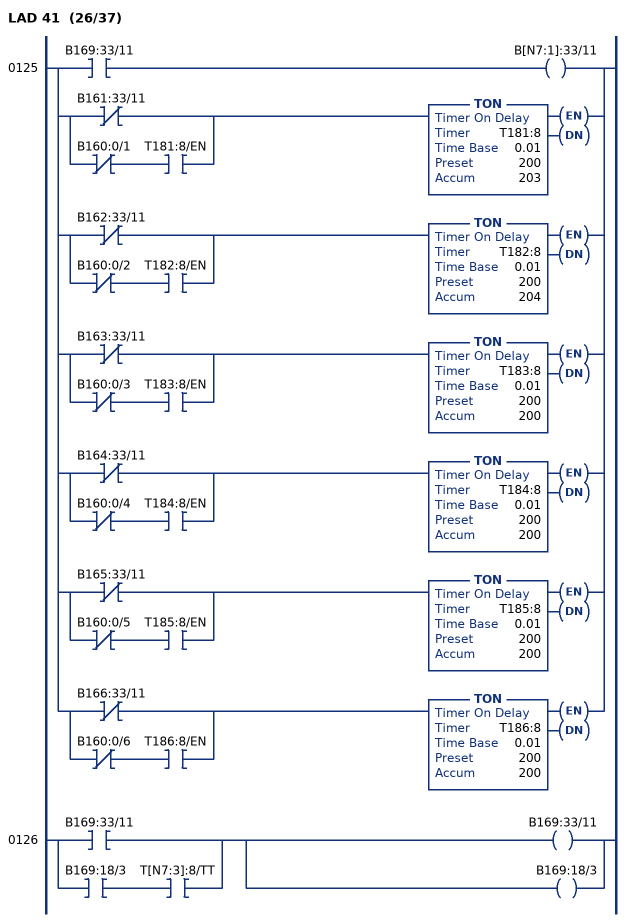
% Rung: 125 %
SOR BST XIC B169:33/11 OTE B[N7:1]:33/11 NXB BST XIO B161:33/11 NXB XIO B160:0/1 XIC T181:8/EN BND TON T181:8 0.01 200 203 NXB BST XIO B162:33/11 NXB XIO B160:0/2 XIC T182:8/EN BND TON T182:8 0.01 200 204 NXB BST XIO B163:33/11 NXB XIO B160:0/3 XIC T183:8/EN BND TON T183:8 0.01 200 200 NXB BST XIO B164:33/11 NXB XIO B160:0/4 XIC T184:8/EN BND TON T184:8 0.01 200 200 NXB BST XIO B165:33/11 NXB XIO B160:0/5 XIC T185:8/EN BND TON T185:8 0.01 200 200 NXB BST XIO B166:33/11 NXB XIO B160:0/6 XIC T186:8/EN BND TON T186:8 0.01 200 200 BND EOR
% Rung: 126 %
SOR BST XIC B169:33/11 NXB XIC B169:18/3 XIC T[N7:3]:8/TT BND BST OTE B169:33/11 NXB OTE B169:18/3 BND EOR

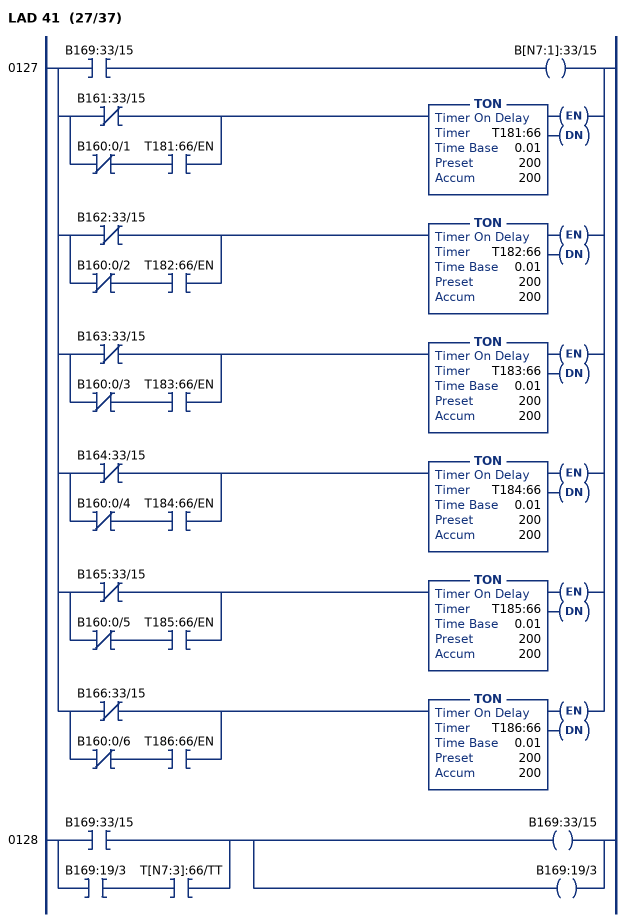
% Rung: 127 %
SOR BST XIC B169:33/15 OTE B[N7:1]:33/15 NXB BST XIO B161:33/15 NXB XIO B160:0/1 XIC T181:66/EN BND TON T181:66 0.01 200 200 NXB BST XIO B162:33/15 NXB XIO B160:0/2 XIC T182:66/EN BND TON T182:66 0.01 200 200 NXB BST XIO B163:33/15 NXB XIO B160:0/3 XIC T183:66/EN BND TON T183:66 0.01 200 200 NXB BST XIO B164:33/15 NXB XIO B160:0/4 XIC T184:66/EN BND TON T184:66 0.01 200 200 NXB BST XIO B165:33/15 NXB XIO B160:0/5 XIC T185:66/EN BND TON T185:66 0.01 200 200 NXB BST XIO B166:33/15 NXB XIO B160:0/6 XIC T186:66/EN BND TON T186:66 0.01 200 200 BND EOR
% Rung: 128 %
SOR BST XIC B169:33/15 NXB XIC B169:19/3 XIC T[N7:3]:66/TT BND BST OTE B169:33/15 NXB OTE B169:19/3 BND EOR

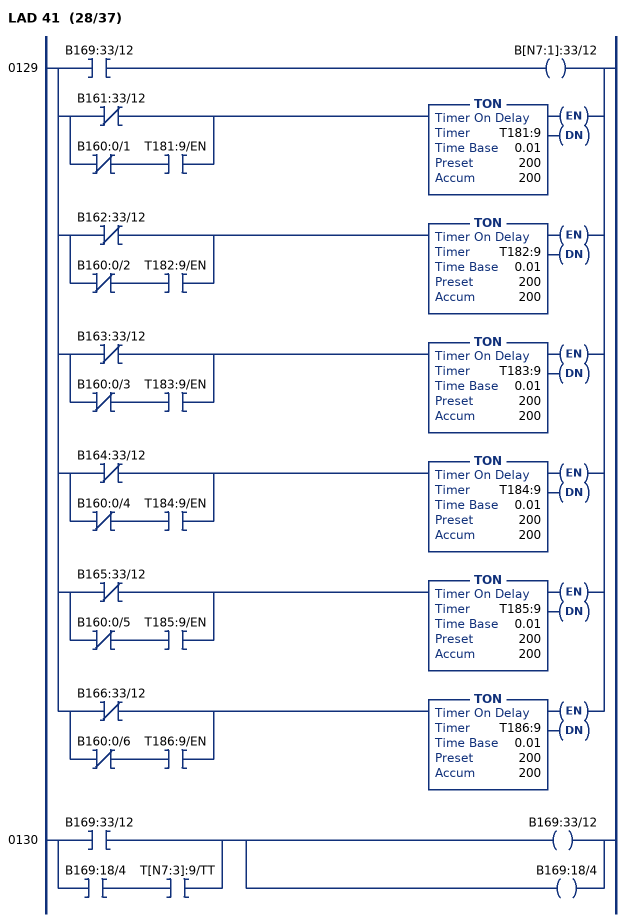
% Rung: 129 %
SOR BST XIC B169:33/12 OTE B[N7:1]:33/12 NXB BST XIO B161:33/12 NXB XIO B160:0/1 XIC T181:9/EN BND TON T181:9 0.01 200 200 NXB BST XIO B162:33/12 NXB XIO B160:0/2 XIC T182:9/EN BND TON T182:9 0.01 200 200 NXB BST XIO B163:33/12 NXB XIO B160:0/3 XIC T183:9/EN BND TON T183:9 0.01 200 200 NXB BST XIO B164:33/12 NXB XIO B160:0/4 XIC T184:9/EN BND TON T184:9 0.01 200 200 NXB BST XIO B165:33/12 NXB XIO B160:0/5 XIC T185:9/EN BND TON T185:9 0.01 200 200 NXB BST XIO B166:33/12 NXB XIO B160:0/6 XIC T186:9/EN BND TON T186:9 0.01 200 200 BND EOR
% Rung: 130 %
SOR BST XIC B169:33/12 NXB XIC B169:18/4 XIC T[N7:3]:9/TT BND BST OTE B169:33/12 NXB OTE B169:18/4 BND EOR

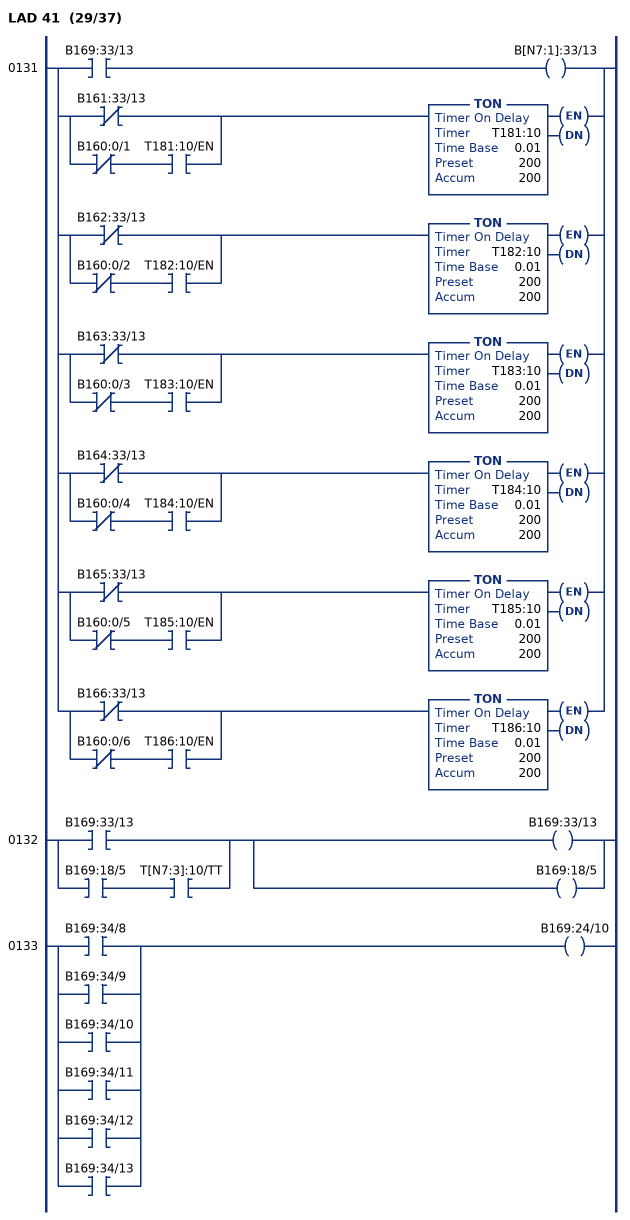
% Rung: 131 %
SOR BST XIC B169:33/13 OTE B[N7:1]:33/13 NXB BST XIO B161:33/13 NXB XIO B160:0/1 XIC T181:10/EN BND TON T181:10 0.01 200 200 NXB BST XIO B162:33/13 NXB XIO B160:0/2 XIC T182:10/EN BND TON T182:10 0.01 200 200 NXB BST XIO B163:33/13 NXB XIO B160:0/3 XIC T183:10/EN BND TON T183:10 0.01 200 200 NXB BST XIO B164:33/13 NXB XIO B160:0/4 XIC T184:10/EN BND TON T184:10 0.01 200 200 NXB BST XIO B165:33/13 NXB XIO B160:0/5 XIC T185:10/EN BND TON T185:10 0.01 200 200 NXB BST XIO B166:33/13 NXB XIO B160:0/6 XIC T186:10/EN BND TON T186:10 0.01 200 200 BND EOR
% Rung: 132 %
SOR BST XIC B169:33/13 NXB XIC B169:18/5 XIC T[N7:3]:10/TT BND BST OTE B169:33/13 NXB OTE B169:18/5 BND EOR
% Rung: 133 %
SOR BST XIC B169:34/8 NXB XIC B169:34/9 NXB XIC B169:34/10 NXB XIC B169:34/11 NXB XIC B169:34/12 NXB XIC B169:34/13 BND OTE B169:24/10 EOR

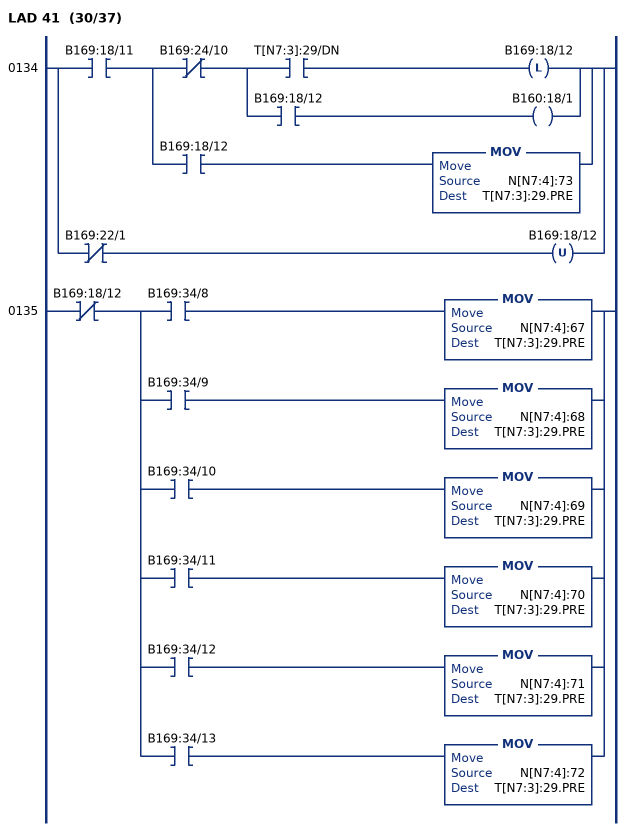
% Rung: 134 %
SOR BST XIC B169:18/11 BST XIO B169:24/10 BST XIC T[N7:3]:29/DN OTL B169:18/12 NXB XIC B169:18/12 OTE B160:18/1 BND NXB XIC B169:18/12 MOV N[N7:4]:73 T[N7:3]:29.PRE BND NXB XIO B169:22/1 OTU B169:18/12 BND EOR
% Rung: 135 %
SOR XIO B169:18/12 BST XIC B169:34/8 MOV N[N7:4]:67 T[N7:3]:29.PRE NXB XIC B169:34/9 MOV N[N7:4]:68 T[N7:3]:29.PRE NXB XIC B169:34/10 MOV N[N7:4]:69 T[N7:3]:29.PRE NXB XIC B169:34/11 MOV N[N7:4]:70 T[N7:3]:29.PRE NXB XIC B169:34/12 MOV N[N7:4]:71 T[N7:3]:29.PRE NXB XIC B169:34/13 MOV N[N7:4]:72 T[N7:3]:29.PRE BND EOR

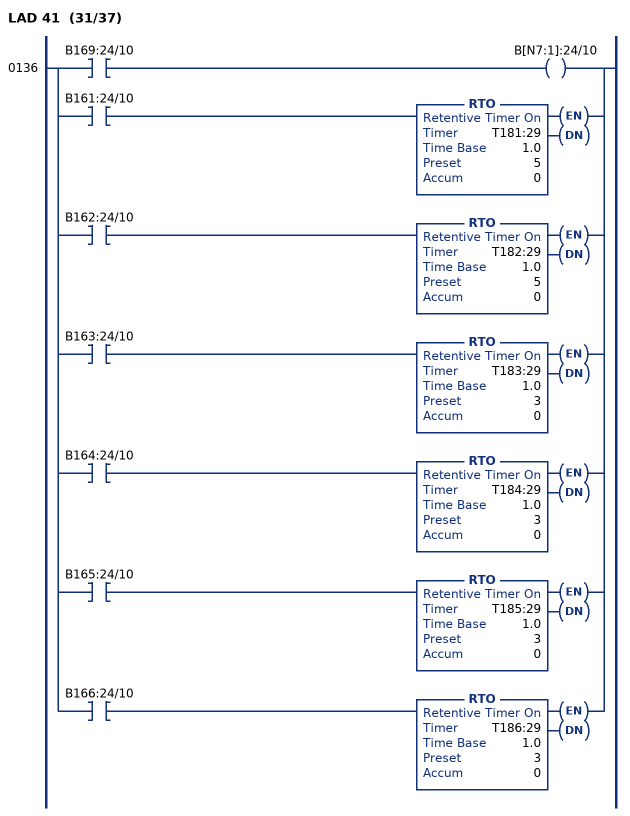
% Rung: 136 %
SOR BST XIC B169:24/10 OTE B[N7:1]:24/10 NXB XIC B161:24/10 RTO T181:29 1.0 5 0 NXB XIC B162:24/10 RTO T182:29 1.0 5 0 NXB XIC B163:24/10 RTO T183:29 1.0 3 0 NXB XIC B164:24/10 RTO T184:29 1.0 3 0 NXB XIC B165:24/10 RTO T185:29 1.0 3 0 NXB XIC B166:24/10 RTO T186:29 1.0 3 0 BND EOR

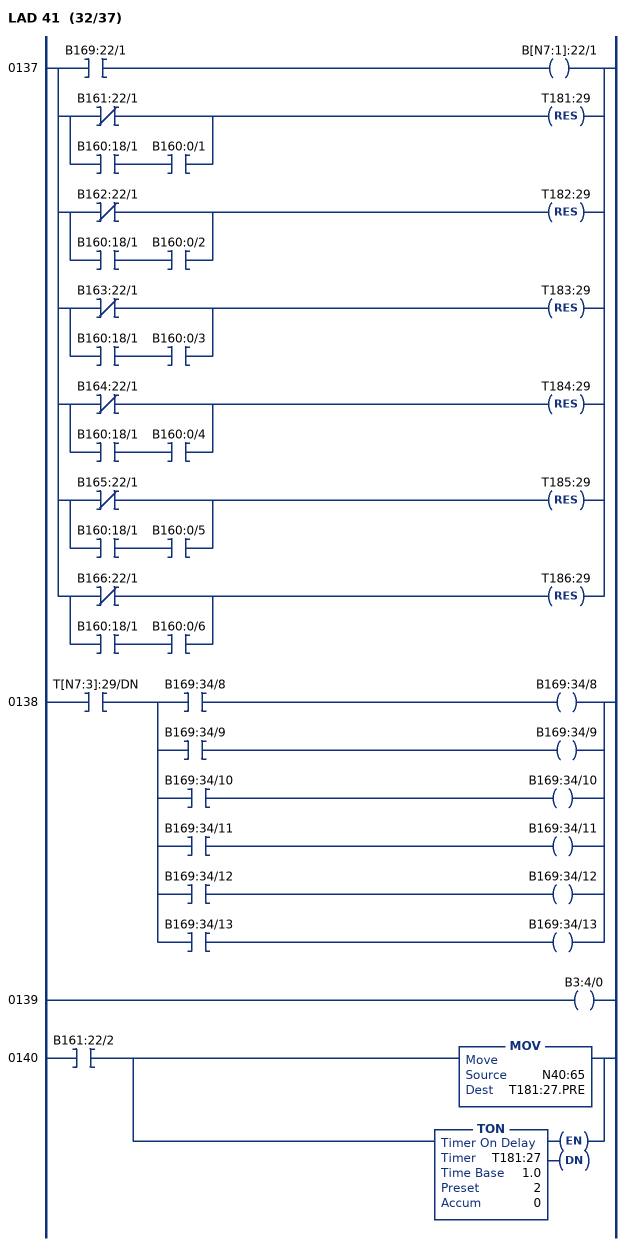
% Rung: 137 %
SOR BST XIC B169:22/1 OTE B[N7:1]:22/1 NXB BST XIO B161:22/1 NXB XIC B160:18/1 XIC B160:0/1 BND RES T181:29 NXB BST XIO B162:22/1 NXB XIC B160:18/1 XIC B160:0/2 BND RES T182:29 NXB BST XIO B163:22/1 NXB XIC B160:18/1 XIC B160:0/3 BND RES T183:29 NXB BST XIO B164:22/1 NXB XIC B160:18/1 XIC B160:0/4 BND RES T184:29 NXB BST XIO B165:22/1 NXB XIC B160:18/1 XIC B160:0/5 BND RES T185:29 NXB BST XIO B166:22/1 NXB XIC B160:18/1 XIC B160:0/6 BND RES T186:29 BND EOR
% Rung: 138 %
SOR XIC T[N7:3]:29/DN BST XIC B169:34/8 OTE B169:34/8 NXB XIC B169:34/9 OTE B169:34/9 NXB XIC B169:34/10 OTE B169:34/10 NXB XIC B169:34/11 OTE B169:34/11 NXB XIC B169:34/12 OTE B169:34/12 NXB XIC B169:34/13 OTE B169:34/13 BND EOR
% Rung: 139 %
SOR OTE B3:4/0 EOR
% Rung: 140 %
SOR XIC B161:22/2 BST MOV N40:65 T181:27.PRE NXB TON T181:27 1.0 2 0 BND EOR

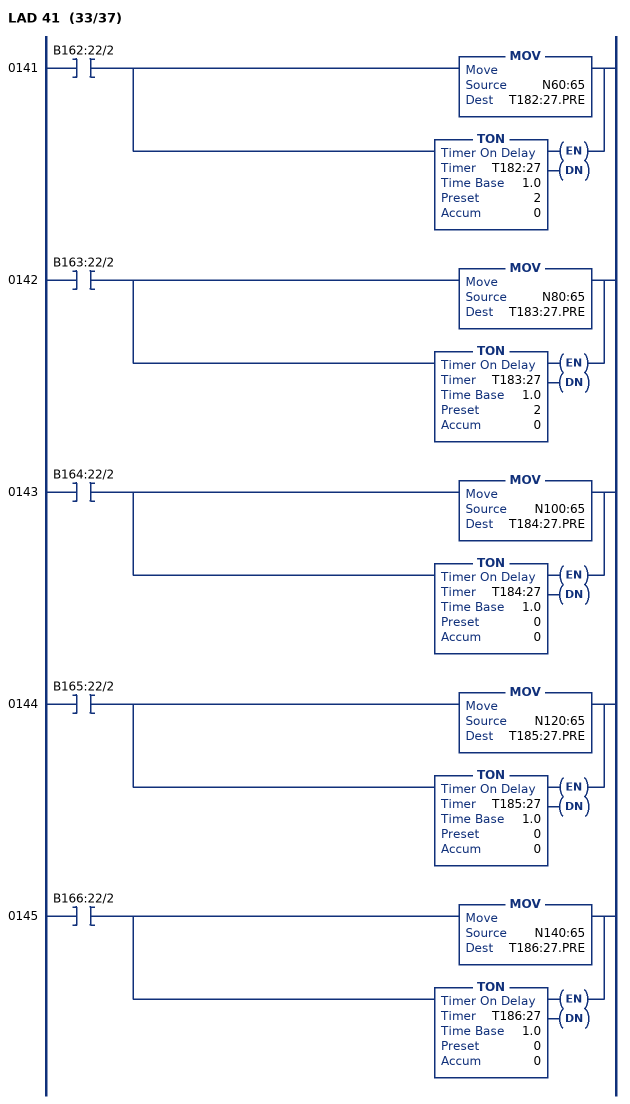
% Rung: 141 %
SOR XIC B162:22/2 BST MOV N60:65 T182:27.PRE NXB TON T182:27 1.0 2 0 BND EOR
% Rung: 142 %
SOR XIC B163:22/2 BST MOV N80:65 T183:27.PRE NXB TON T183:27 1.0 2 0 BND EOR
% Rung: 143 %
SOR XIC B164:22/2 BST MOV N100:65 T184:27.PRE NXB TON T184:27 1.0 0 0 BND EOR
% Rung: 144 %
SOR XIC B165:22/2 BST MOV N120:65 T185:27.PRE NXB TON T185:27 1.0 0 0 BND EOR
% Rung: 145 %
SOR XIC B166:22/2 BST MOV N140:65 T186:27.PRE NXB TON T186:27 1.0 0 0 BND EOR

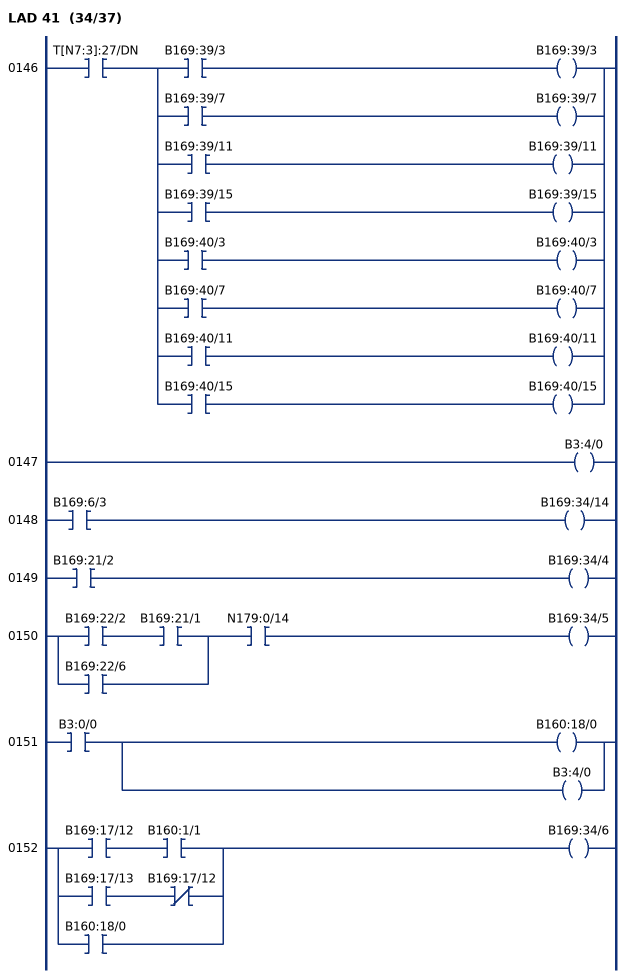
% Rung: 146 %
SOR XIC T[N7:3]:27/DN BST XIC B169:39/3 OTE B169:39/3 NXB XIC B169:39/7 OTE B169:39/7 NXB XIC B169:39/11 OTE B169:39/11 NXB XIC B169:39/15 OTE B169:39/15 NXB XIC B169:40/3 OTE B169:40/3 NXB XIC B169:40/7 OTE B169:40/7 NXB XIC B169:40/11 OTE B169:40/11 NXB XIC B169:40/15 OTE B169:40/15 BND EOR
% Rung: 147 %
SOR OTE B3:4/0 EOR
% Rung: 148 %
SOR XIC B169:6/3 OTE B169:34/14 EOR
% Rung: 149 %
SOR XIC B169:21/2 OTE B169:34/4 EOR
% Rung: 150 %
SOR BST XIC B169:22/2 XIC B169:21/1 NXB XIC B169:22/6 BND XIC N179:0/14 OTE B169:34/5 EOR
% Rung: 151 %
SOR XIC B3:0/0 BST OTE B160:18/0 NXB OTE B3:4/0 BND EOR
% Rung: 152 %
SOR BST XIC B169:17/12 XIC B160:1/1 NXB XIC B169:17/13 XIO B169:17/12 NXB XIC B160:18/0 BND OTE B169:34/6 EOR

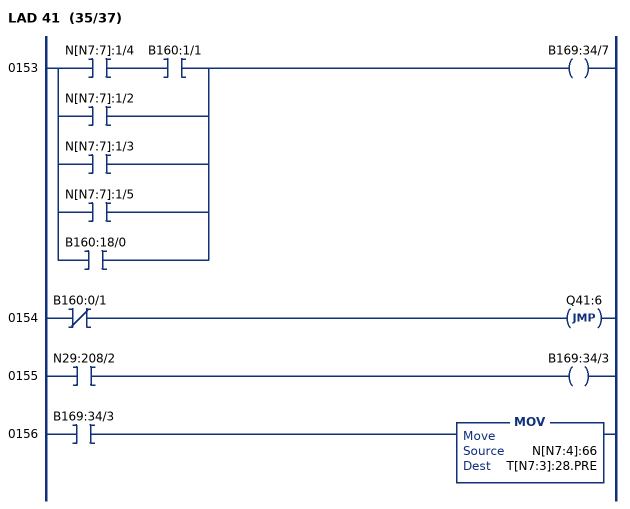
% Rung: 153 %
SOR BST XIC N[N7:7]:1/4 XIC B160:1/1 NXB XIC N[N7:7]:1/2 NXB XIC N[N7:7]:1/3 NXB XIC N[N7:7]:1/5 NXB XIC B160:18/0 BND OTE B169:34/7 EOR
% Rung: 154 %
SOR XIO B160:0/1 JMP Q41:6 EOR
% Rung: 155 %
SOR XIC N29:208/2 OTE B169:34/3 EOR
% Rung: 156 %
SOR XIC B169:34/3 MOV N[N7:4]:66 T[N7:3]:28.PRE EOR

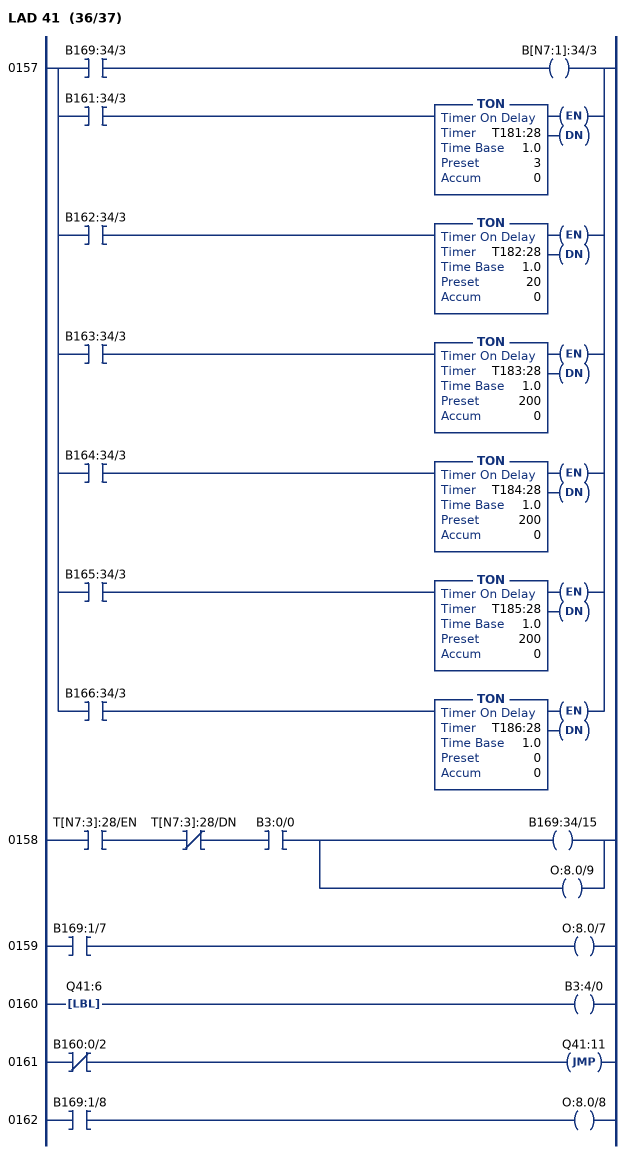
% Rung: 157 %
SOR BST XIC B169:34/3 OTE B[N7:1]:34/3 NXB XIC B161:34/3 TON T181:28 1.0 3 0 NXB XIC B162:34/3 TON T182:28 1.0 20 0 NXB XIC B163:34/3 TON T183:28 1.0 200 0 NXB XIC B164:34/3 TON T184:28 1.0 200 0 NXB XIC B165:34/3 TON T185:28 1.0 200 0 NXB XIC B166:34/3 TON T186:28 1.0 0 0 BND EOR
% Rung: 158 %
SOR XIC T[N7:3]:28/EN XIO T[N7:3]:28/DN XIC B3:0/0 BST OTE B169:34/15 NXB OTE O:8.0/9 BND EOR
% Rung: 159 %
SOR XIC B169:1/7 OTE O:8.0/7 EOR
% Rung: 160 %
SOR LBL Q41:6 OTE B3:4/0 EOR
% Rung: 161 %
SOR XIO B160:0/2 JMP Q41:11 EOR
% Rung: 162 %
SOR XIC B169:1/8 OTE O:8.0/8 EOR

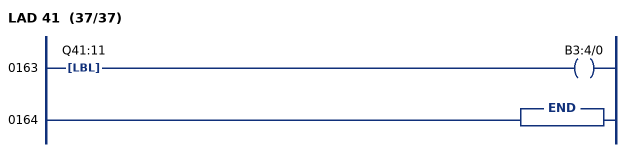
% Rung: 163 %
SOR LBL Q41:11 OTE B3:4/0 EOR
% Rung: 164 %
SOR END EOR

LADDER 42
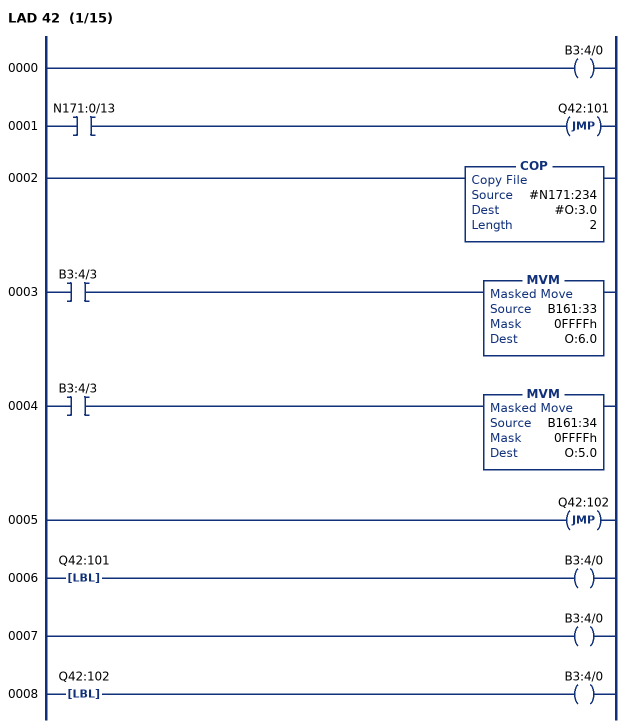
% Rung: 0 %
SOR OTE B3:4/0 EOR
% Rung: 1 %
SOR XIC N171:0/13 JMP Q42:101 EOR
% Rung: 2 %
SOR COP #N171:234 #O:3.0 2 EOR
% Rung: 3 %
SOR XIC B3:4/3 MVM B161:33 0FFFFh O:6.0 EOR
% Rung: 4 %
SOR XIC B3:4/3 MVM B161:34 0FFFFh O:5.0 EOR
% Rung: 5 %
SOR JMP Q42:102 EOR
% Rung: 6 %
SOR LBL Q42:101 OTE B3:4/0 EOR
% Rung: 7 %
SOR OTE B3:4/0 EOR
% Rung: 8 %
SOR LBL Q42:102 OTE B3:4/0 EOR

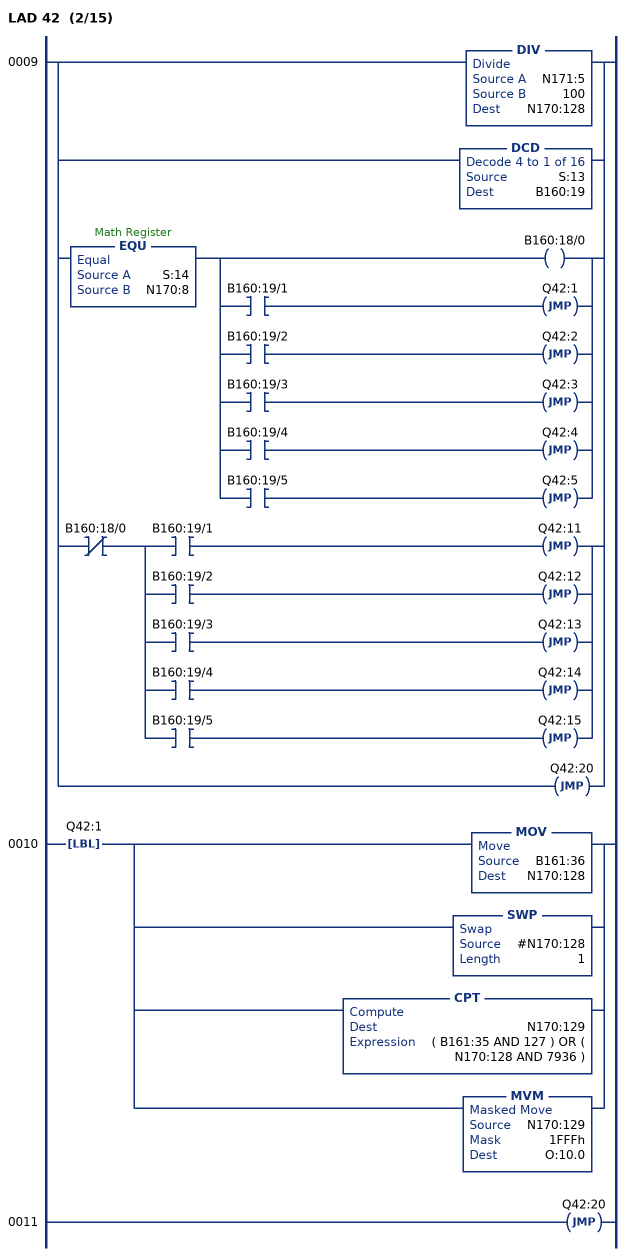
% Rung: 9 %
SOR BST DIV N171:5 100 N170:128 NXB DCD S:13 B160:19 NXB EQU S:14 N170:8 BST OTE B160:18/0 NXB XIC B160:19/1 JMP Q42:1 NXB XIC B160:19/2 JMP Q42:2 NXB XIC B160:19/3 JMP Q42:3 NXB XIC B160:19/4 JMP Q42:4 NXB XIC B160:19/5 JMP Q42:5 BND NXB XIO B160:18/0 BST XIC B160:19/1 JMP Q42:11 NXB XIC B160:19/2 JMP Q42:12 NXB XIC B160:19/3 JMP Q42:13 NXB XIC B160:19/4 JMP Q42:14 NXB XIC B160:19/5 JMP Q42:15 BND NXB JMP Q42:20 BND EOR
%   S:13  "Math Register" %
%   S:14  "Math Register" %
% Rung: 10 %
SOR LBL Q42:1 BST MOV B161:36 N170:128 NXB SWP #N170:128 1 NXB CPT N170:129 " ( B161:35 AND 127 ) OR ( N170:128 AND 7936 ) " NXB MVM N170:129 1FFFh O:10.0 BND EOR
% Rung: 11 %
SOR JMP Q42:20 EOR

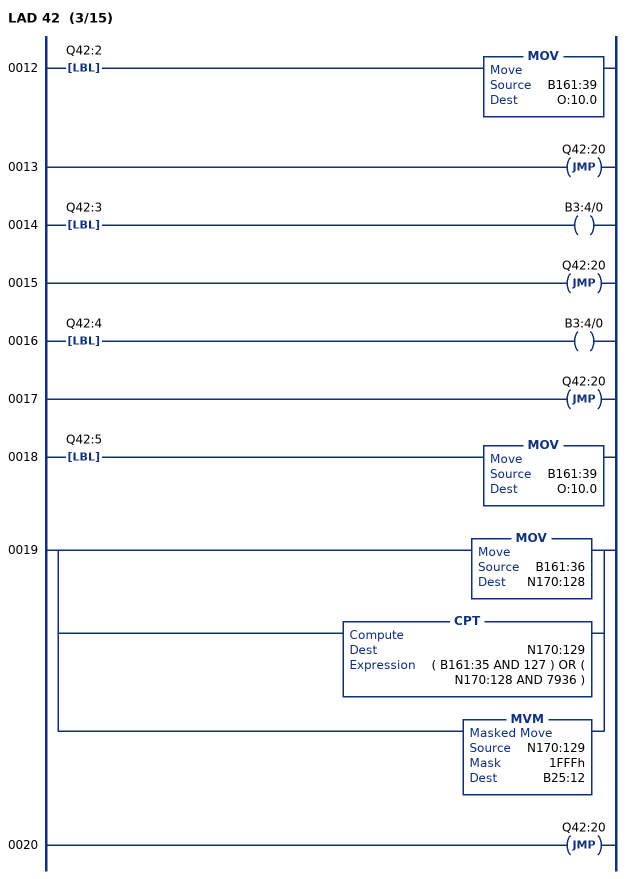
% Rung: 12 %
SOR LBL Q42:2 MOV B161:39 O:10.0 EOR
% Rung: 13 %
SOR JMP Q42:20 EOR
% Rung: 14 %
SOR LBL Q42:3 OTE B3:4/0 EOR
% Rung: 15 %
SOR JMP Q42:20 EOR
% Rung: 16 %
SOR LBL Q42:4 OTE B3:4/0 EOR
% Rung: 17 %
SOR JMP Q42:20 EOR
% Rung: 18 %
SOR LBL Q42:5 MOV B161:39 O:10.0 EOR
% Rung: 19 %
SOR BST MOV B161:36 N170:128 NXB CPT N170:129 " ( B161:35 AND 127 ) OR ( N170:128 AND 7936 ) " NXB MVM N170:129 1FFFh B25:12 BND EOR
% Rung: 20 %
SOR JMP Q42:20 EOR

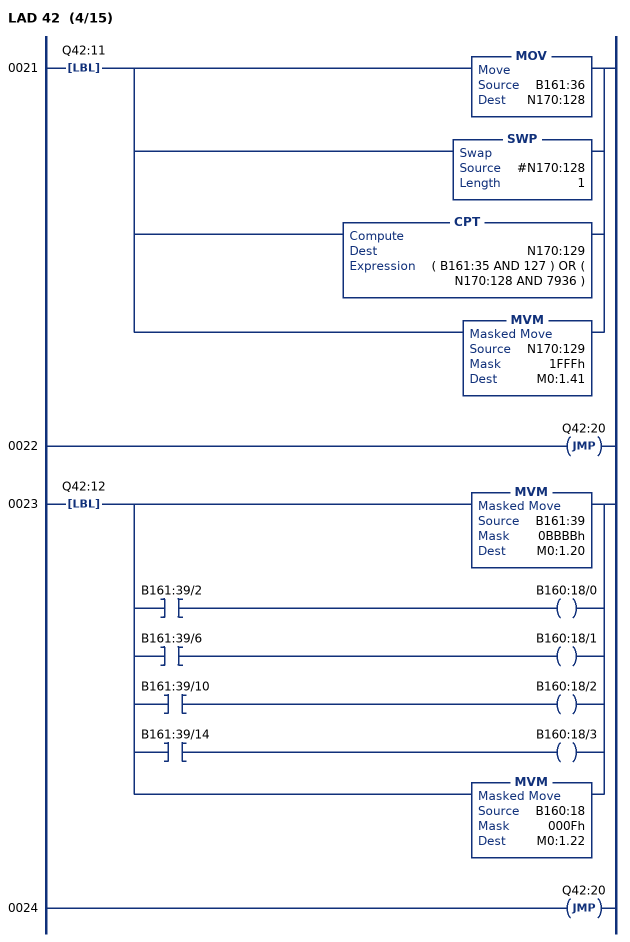
% Rung: 21 %
SOR LBL Q42:11 BST MOV B161:36 N170:128 NXB SWP #N170:128 1 NXB CPT N170:129 " ( B161:35 AND 127 ) OR ( N170:128 AND 7936 ) " NXB MVM N170:129 1FFFh M0:1.41 BND EOR
% Rung: 22 %
SOR JMP Q42:20 EOR
% Rung: 23 %
SOR LBL Q42:12 BST MVM B161:39 0BBBBh M0:1.20 NXB XIC B161:39/2 OTE B160:18/0 NXB XIC B161:39/6 OTE B160:18/1 NXB XIC B161:39/10 OTE B160:18/2 NXB XIC B161:39/14 OTE B160:18/3 NXB MVM B160:18 000Fh M0:1.22 BND EOR
% Rung: 24 %
SOR JMP Q42:20 EOR

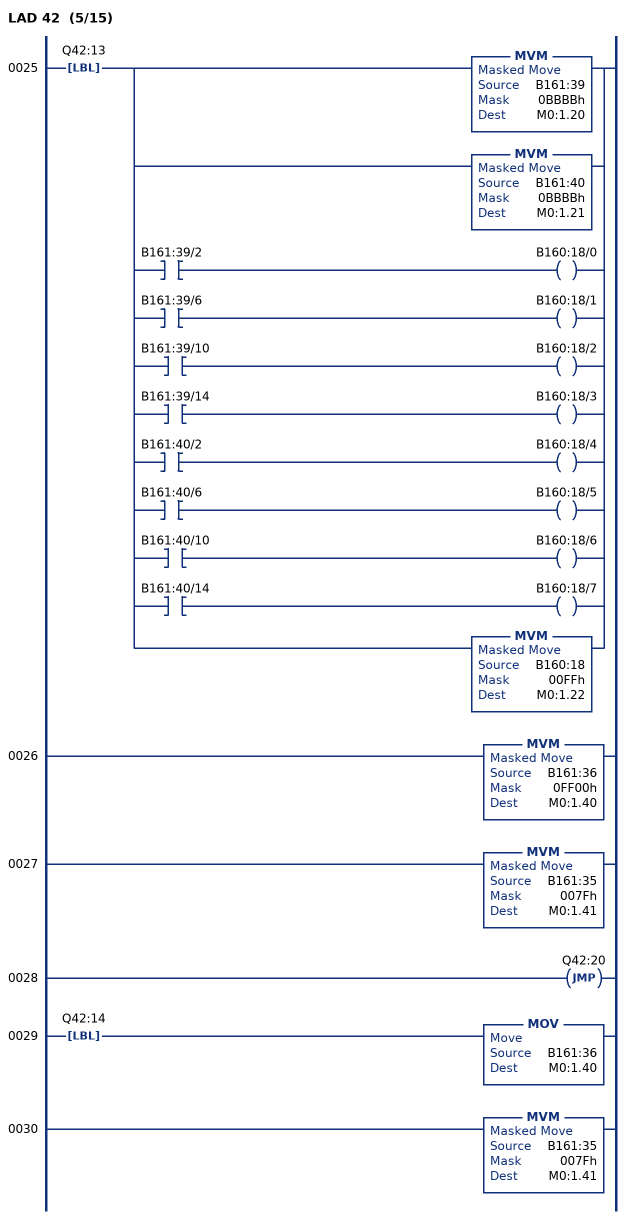
% Rung: 25 %
SOR LBL Q42:13 BST MVM B161:39 0BBBBh M0:1.20 NXB MVM B161:40 0BBBBh M0:1.21 NXB XIC B161:39/2 OTE B160:18/0 NXB XIC B161:39/6 OTE B160:18/1 NXB XIC B161:39/10 OTE B160:18/2 NXB XIC B161:39/14 OTE B160:18/3 NXB XIC B161:40/2 OTE B160:18/4 NXB XIC B161:40/6 OTE B160:18/5 NXB XIC B161:40/10 OTE B160:18/6 NXB XIC B161:40/14 OTE B160:18/7 NXB MVM B160:18 00FFh M0:1.22 BND EOR
% Rung: 26 %
SOR MVM B161:36 0FF00h M0:1.40 EOR
% Rung: 27 %
SOR MVM B161:35 007Fh M0:1.41 EOR
% Rung: 28 %
SOR JMP Q42:20 EOR
% Rung: 29 %
SOR LBL Q42:14 MOV B161:36 M0:1.40 EOR
% Rung: 30 %
SOR MVM B161:35 007Fh M0:1.41 EOR

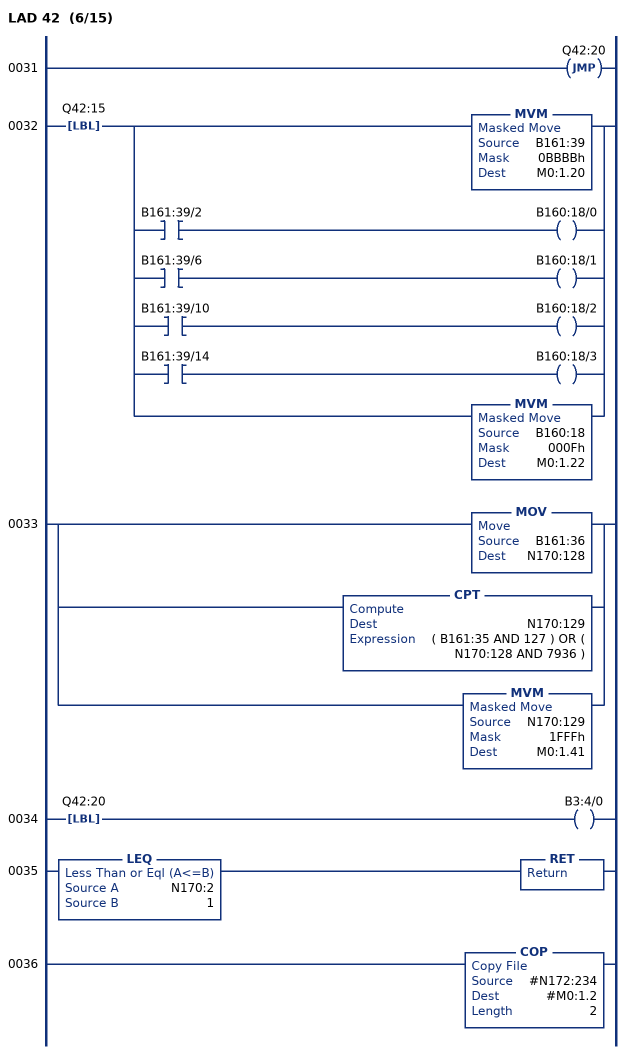
% Rung: 31 %
SOR JMP Q42:20 EOR
% Rung: 32 %
SOR LBL Q42:15 BST MVM B161:39 0BBBBh M0:1.20 NXB XIC B161:39/2 OTE B160:18/0 NXB XIC B161:39/6 OTE B160:18/1 NXB XIC B161:39/10 OTE B160:18/2 NXB XIC B161:39/14 OTE B160:18/3 NXB MVM B160:18 000Fh M0:1.22 BND EOR
% Rung: 33 %
SOR BST MOV B161:36 N170:128 NXB CPT N170:129 " ( B161:35 AND 127 ) OR ( N170:128 AND 7936 ) " NXB MVM N170:129 1FFFh M0:1.41 BND EOR
% Rung: 34 %
SOR LBL Q42:20 OTE B3:4/0 EOR
% Rung: 35 %
SOR LEQ N170:2 1 RET EOR
% Rung: 36 %
SOR COP #N172:234 #M0:1.2 2 EOR

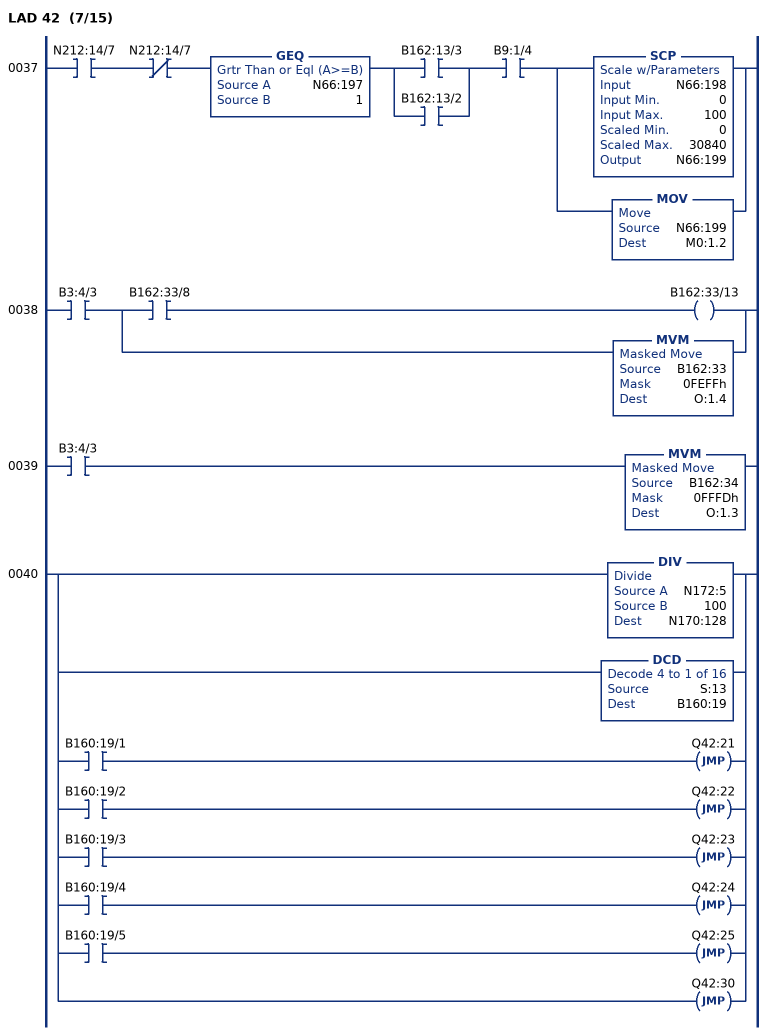
% Rung: 37 %
SOR XIC N212:14/7 XIO N212:14/7 GEQ N66:197 1 BST XIC B162:13/3 NXB XIC B162:13/2 BND XIC B9:1/4 BST SCP N66:198 0 100 0 30840 N66:199 NXB MOV N66:199 M0:1.2 BND EOR
% Rung: 38 %
SOR XIC B3:4/3 BST XIC B162:33/8 OTE B162:33/13 NXB MVM B162:33 0FEFFh O:1.4 BND EOR
% Rung: 39 %
SOR XIC B3:4/3 MVM B162:34 0FFFDh O:1.3 EOR
% Rung: 40 %
SOR BST DIV N172:5 100 N170:128 NXB DCD S:13 B160:19 NXB BST XIC B160:19/1 JMP Q42:21 NXB XIC B160:19/2 JMP Q42:22 NXB XIC B160:19/3 JMP Q42:23 NXB XIC B160:19/4 JMP Q42:24 NXB XIC B160:19/5 JMP Q42:25 BND NXB JMP Q42:30 BND EOR
%   S:13  "Math Register" %

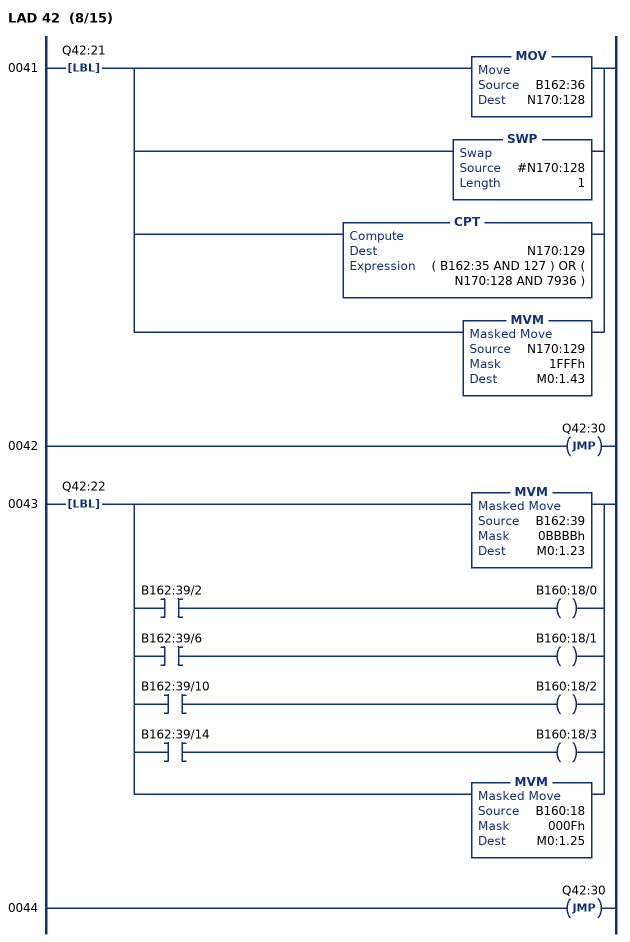
% Rung: 41 %
SOR LBL Q42:21 BST MOV B162:36 N170:128 NXB SWP #N170:128 1 NXB CPT N170:129 " ( B162:35 AND 127 ) OR ( N170:128 AND 7936 ) " NXB MVM N170:129 1FFFh M0:1.43 BND EOR
% Rung: 42 %
SOR JMP Q42:30 EOR
% Rung: 43 %
SOR LBL Q42:22 BST MVM B162:39 0BBBBh M0:1.23 NXB XIC B162:39/2 OTE B160:18/0 NXB XIC B162:39/6 OTE B160:18/1 NXB XIC B162:39/10 OTE B160:18/2 NXB XIC B162:39/14 OTE B160:18/3 NXB MVM B160:18 000Fh M0:1.25 BND EOR
% Rung: 44 %
SOR JMP Q42:30 EOR

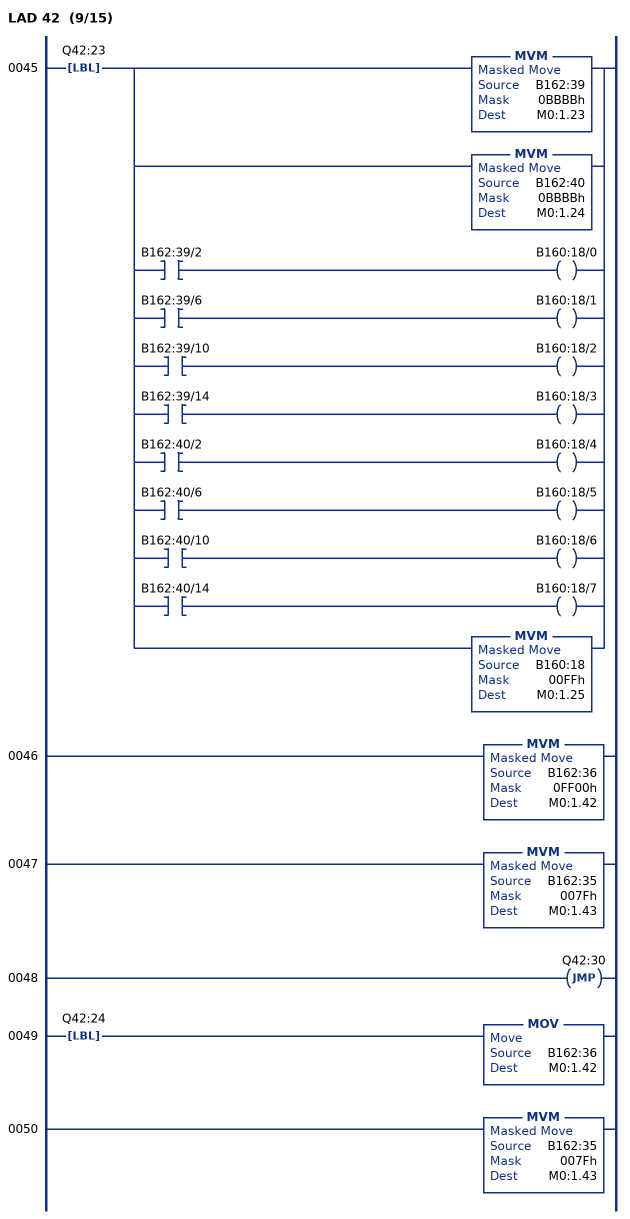
% Rung: 45 %
SOR LBL Q42:23 BST MVM B162:39 0BBBBh M0:1.23 NXB MVM B162:40 0BBBBh M0:1.24 NXB XIC B162:39/2 OTE B160:18/0 NXB XIC B162:39/6 OTE B160:18/1 NXB XIC B162:39/10 OTE B160:18/2 NXB XIC B162:39/14 OTE B160:18/3 NXB XIC B162:40/2 OTE B160:18/4 NXB XIC B162:40/6 OTE B160:18/5 NXB XIC B162:40/10 OTE B160:18/6 NXB XIC B162:40/14 OTE B160:18/7 NXB MVM B160:18 00FFh M0:1.25 BND EOR
% Rung: 46 %
SOR MVM B162:36 0FF00h M0:1.42 EOR
% Rung: 47 %
SOR MVM B162:35 007Fh M0:1.43 EOR
% Rung: 48 %
SOR JMP Q42:30 EOR
% Rung: 49 %
SOR LBL Q42:24 MOV B162:36 M0:1.42 EOR
% Rung: 50 %
SOR MVM B162:35 007Fh M0:1.43 EOR

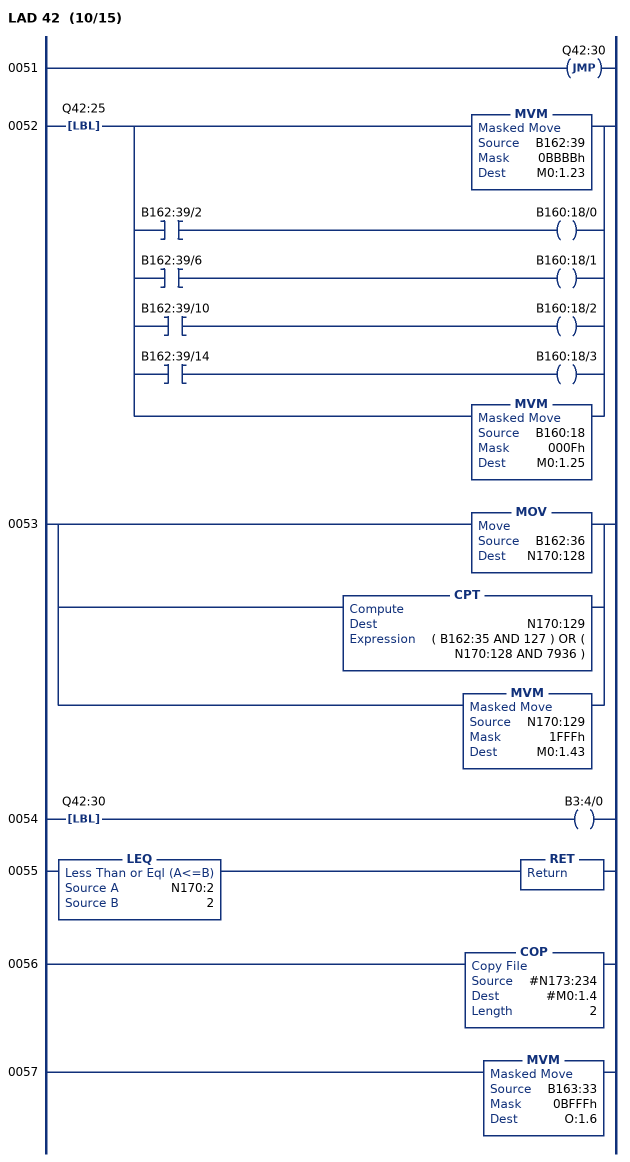
% Rung: 51 %
SOR JMP Q42:30 EOR
% Rung: 52 %
SOR LBL Q42:25 BST MVM B162:39 0BBBBh M0:1.23 NXB XIC B162:39/2 OTE B160:18/0 NXB XIC B162:39/6 OTE B160:18/1 NXB XIC B162:39/10 OTE B160:18/2 NXB XIC B162:39/14 OTE B160:18/3 NXB MVM B160:18 000Fh M0:1.25 BND EOR
% Rung: 53 %
SOR BST MOV B162:36 N170:128 NXB CPT N170:129 " ( B162:35 AND 127 ) OR ( N170:128 AND 7936 ) " NXB MVM N170:129 1FFFh M0:1.43 BND EOR
% Rung: 54 %
SOR LBL Q42:30 OTE B3:4/0 EOR
% Rung: 55 %
SOR LEQ N170:2 2 RET EOR
% Rung: 56 %
SOR COP #N173:234 #M0:1.4 2 EOR
% Rung: 57 %
SOR MVM B163:33 0BFFFh O:1.6 EOR

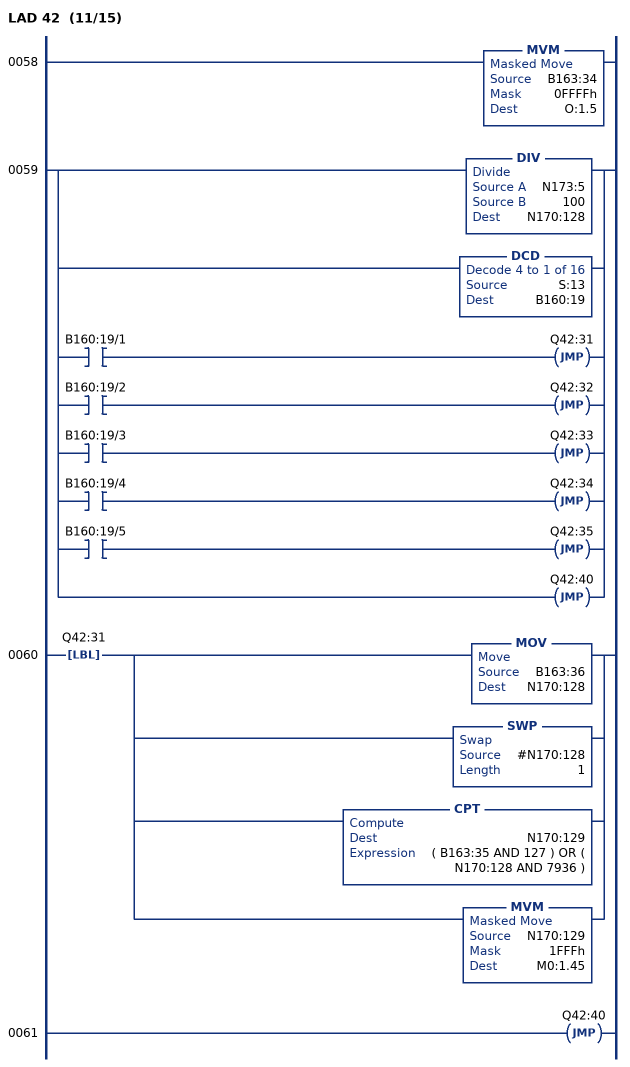
% Rung: 58 %
SOR MVM B163:34 0FFFFh O:1.5 EOR
% Rung: 59 %
SOR BST DIV N173:5 100 N170:128 NXB DCD S:13 B160:19 NXB BST XIC B160:19/1 JMP Q42:31 NXB XIC B160:19/2 JMP Q42:32 NXB XIC B160:19/3 JMP Q42:33 NXB XIC B160:19/4 JMP Q42:34 NXB XIC B160:19/5 JMP Q42:35 BND NXB JMP Q42:40 BND EOR
%   S:13  "Math Register" %
% Rung: 60 %
SOR LBL Q42:31 BST MOV B163:36 N170:128 NXB SWP #N170:128 1 NXB CPT N170:129 " ( B163:35 AND 127 ) OR ( N170:128 AND 7936 ) " NXB MVM N170:129 1FFFh M0:1.45 BND EOR
% Rung: 61 %
SOR JMP Q42:40 EOR

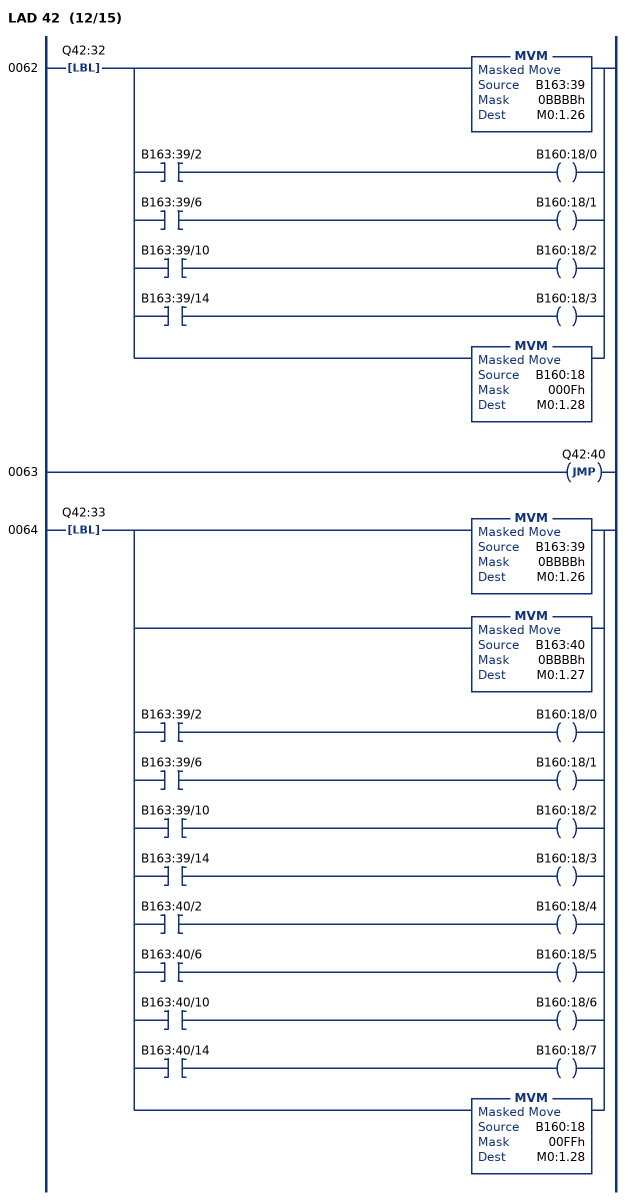
% Rung: 62 %
SOR LBL Q42:32 BST MVM B163:39 0BBBBh M0:1.26 NXB XIC B163:39/2 OTE B160:18/0 NXB XIC B163:39/6 OTE B160:18/1 NXB XIC B163:39/10 OTE B160:18/2 NXB XIC B163:39/14 OTE B160:18/3 NXB MVM B160:18 000Fh M0:1.28 BND EOR
% Rung: 63 %
SOR JMP Q42:40 EOR
% Rung: 64 %
SOR LBL Q42:33 BST MVM B163:39 0BBBBh M0:1.26 NXB MVM B163:40 0BBBBh M0:1.27 NXB XIC B163:39/2 OTE B160:18/0 NXB XIC B163:39/6 OTE B160:18/1 NXB XIC B163:39/10 OTE B160:18/2 NXB XIC B163:39/14 OTE B160:18/3 NXB XIC B163:40/2 OTE B160:18/4 NXB XIC B163:40/6 OTE B160:18/5 NXB XIC B163:40/10 OTE B160:18/6 NXB XIC B163:40/14 OTE B160:18/7 NXB MVM B160:18 00FFh M0:1.28 BND EOR

